FUNCTION_BLOCK MSb (* Basic FB with empty ECC *)
  (* Standard: 61499-2 *)
  (* Version 1.0, 0000-00-00, 0 *)
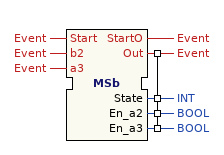
  EVENT_INPUT
    Start;
    b2;
    a3;
  END_EVENT
  EVENT_OUTPUT
    StartO;
    Out WITH State, En_a2, En_a3;
  END_EVENT
  VAR_OUTPUT
    State : INT := 1;
    En_a2 : BOOL := 1;
    En_a3 : BOOL := 1;
  END_VAR
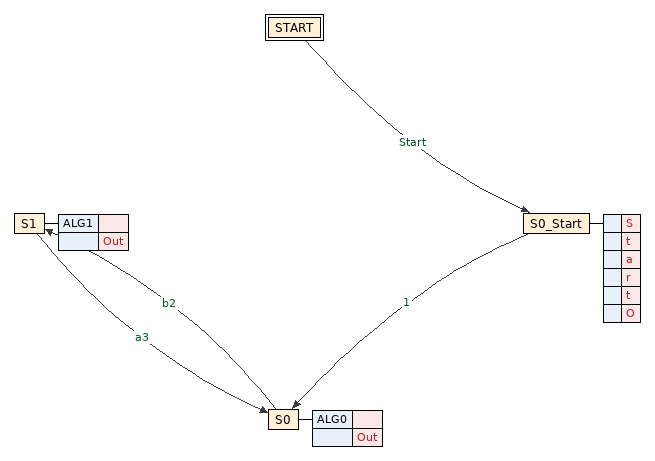
  EC_STATES
    START; (* Initial State *)
    S0_Start : -> S, -> t, -> a, -> r, -> t, -> O;
    S0 : ALG0, -> Out;
    S1 : ALG1, -> Out;
  END_STATES
  EC_TRANSITIONS
    START TO S0_Start := Start;
    S0_Start TO S0 := 1;
    S0 TO S1 := b2;
    S1 TO S0 := a3;
  END_TRANSITIONS
  ALGORITHM ALG0 IN ST:
State:=0;
				En_a2:=True;
				En_a3:=False;
  END_ALGORITHM
  ALGORITHM ALG1 IN ST:
State:=1;
				En_a2:=False;
				En_a3:=True;
  END_ALGORITHM
END_FUNCTION_BLOCK
